{attribute 'qualified_only'}
VAR_GLOBAL
	bAutoMan : SR;
END_VAR

(* stored: Version 1.1.0.1, ProductVersion 3.1.4024.12
   GVL Tags: Id {c5a4b9f5-18a7-4af3-9463-d2c265e7bcc5} *)
